FUNCTION_BLOCK FB_InfeedFoodUnit EXTENDS FB_BaseMainStation
VAR_INPUT
END_VAR
VAR_OUTPUT
END_VAR
VAR	
	{ attribute 'TcHmiSystemEng.Parameter.Name' := 'Cut Cylinder' }
	_fbCutCylinder			: FB_Cylinder;
END_VAR

END_FUNCTION_BLOCK

(* stored: Version 1.1.0.1
   POU FB_InfeedFoodUnit: Id {4afe9da4-120b-4ce2-9b40-91ba1a4ebb78}, SpecialFunc None *)
